{attribute 'qualified_only'}
{attribute 'strict'}
{attribute 'to_string'}
TYPE nGechterPress_ErrorCodes :
(
	// Błędy ogólne
	NoError := 0,
	UnKnownAlarm := 53,						// Niezidentyfikowany alarm maszyny
	UnKnownLock := 54,						// Niezidentyfikowana blokada maszyny
	ProgramConfigError := 90,				// Błąd w konfiguracji programu
	ResetTimeout := 518,					// Timeout resetu maszyny
	SafetySystemNotArmed := 614,			// System safety nie uzbrojony
	NoMachineReactionOnStartSig := 140,		// Brak reakcji na sygnał startu (brak wysunięcia siłownika - brak powietrza itp.)
	TwoHandStartReleasedToEarly := 96,		// Dwustart zwolniony zbyt wcześnie
	
	OperInteruptedBeforeWorkPos := 132,		// Za wcześnie puszczono dwustart - część nie wprasowana
	ToLowAirPressure	:= 290,				// Niskie ciśnienie sprężonego powietrza 
	PressPossitionMeasureError := 291		// Błąd pomiaru pozycji prasy
);
END_TYPE

(* stored: Version 1.1.0.1, ProductVersion 3.1.4024.12
   EnumerationTextList nGechterPress_ErrorCodes: Id {84f4f40e-f3d6-4b88-914b-9854b1b56523} *)
